{attribute 'linkalways'} 
{attribute 'no_explicit_call' := 'This FB is a CLASS and must be accessed using methods or properties'}
{attribute 'enable_dynamic_creation'}
FUNCTION_BLOCK Node_F_VN_SubtractScalarFromImage EXTENDS VisionNode
VAR
    ipSrcImage : _ITcVnImage;
    fScalar : _LREAL(0.0);
    ipDestImage : _ITcVnImage;
    hrPrev : _HRESULT(S_OK);
	hresult : _HRESULT(S_OK);
END_VAR

METHOD PUBLIC  Clone : I_Node
VAR
	pNode : POINTER TO Node_F_VN_SubtractScalarFromImage;
END_VAR
pNode := __NEW(Node_F_VN_SubtractScalarFromImage);
Clone := pNode^;
END_METHOD

METHOD FB_init : BOOL
VAR_INPUT
	bInitRetains : BOOL; // if TRUE, the retain variables are initialized (warm start / cold start)
	bInCopyCode : BOOL;  // if TRUE, the instance afterwards gets moved into the copy code (online change)
END_VAR
AddInput('ipSrcImage', ipSrcImage);
AddInput('fScalar', fScalar);
AddInput('hrPrev', hrPrev);
AddOutput('ipDestImage', ipDestImage);
AddOutput('hresult',hresult);
END_METHOD

METHOD PROTECTED OnExecute : HRESULT
hresult.Value := F_VN_SubtractScalarFromImage(
    ipSrcImage := ipSrcImage.Value,
    fScalar := fScalar.Value,
	ipDestImage := ipDestImage.Value,
	hrPrev:= hrPrev.Value);
END_METHOD

METHOD PUBLIC PreExecutionCheck
VAR_INPUT
	Check : I_PreExecutionChecks;
END_VAR
IF FAILED(hrPrev.Value) THEN
    RETURN;
END_IF

Check.IsTrue(ipSrcImage.IsValid, 'ipSrcImage must contain an image');
END_METHOD

END_FUNCTION_BLOCK

(* stored: Version 1.1.0.1, ProductVersion 3.1.4024.13
   POU Node_F_VN_SubtractScalarFromImage: Id {37eff8c5-098d-04a6-26d4-b3929c28010f}, SpecialFunc None
   Folder Constructor: Id {386ace35-a85d-0b6e-030f-86de042c6551}
   Method Clone: Id {7be79408-aa72-0cb2-214b-764110e41dda}
   Method FB_init: Id {934f30c6-7172-0ded-056e-4dc04589f6b0}
   Method OnExecute: Id {a13c82e6-a903-0ced-16f2-78d8a28b5fe8}
   Method PreExecutionCheck: Id {831443b7-4a08-09a1-3b6e-31c703996a83} *)
